// TIA Portal V21 export
DATA_BLOCK "DB623"   // DB623
TITLE = DB618
{ S7_Optimized_Access := 'FALSE' }
// Recipe
// stored: AutoNumber false
   VAR RETAIN
      StepEnable : Array[0..5] of Bool;
      Mm01Speed : Real := 1200.0;
      Cp01Speed : Real := 1000.0;
      DrainPressure : Real := 1.11;
      AirPurgingPressure : Real := 1.33;
      SystemDrainTime : Int := 30;
      PreRinseCycleSelection : Int := 1;
      FillingCycleSelection : Int := 1;
      FinalRinseCycleSelection : Int := 1;
      PreRinseCycleNoOfRep : Int := 1;
      FillingCycleNoOfRep : Int := 2;
      FillingCycleMixingTime : Int := 30;
      FinalRinseCycleMixingTime : Int := 35;
      FillingCycleFillQty : Real := 500.0;
      FinalRinseCycleFillQty : Real := 1000.0;
      PreRinseCycleSelString : String[10];
      FillingCycleSelString : String[10];
      FinalRinseCycleSelString : String[10];
      FinalRinseSetCond : Real := 1.22;
      SbiOnTime : Int := 10;
      SbiOffTime : Int := 5;
   END_VAR
BEGIN
   StepEnable[0] := FALSE;
   StepEnable[1..3] := TRUE;
END_DATA_BLOCK
